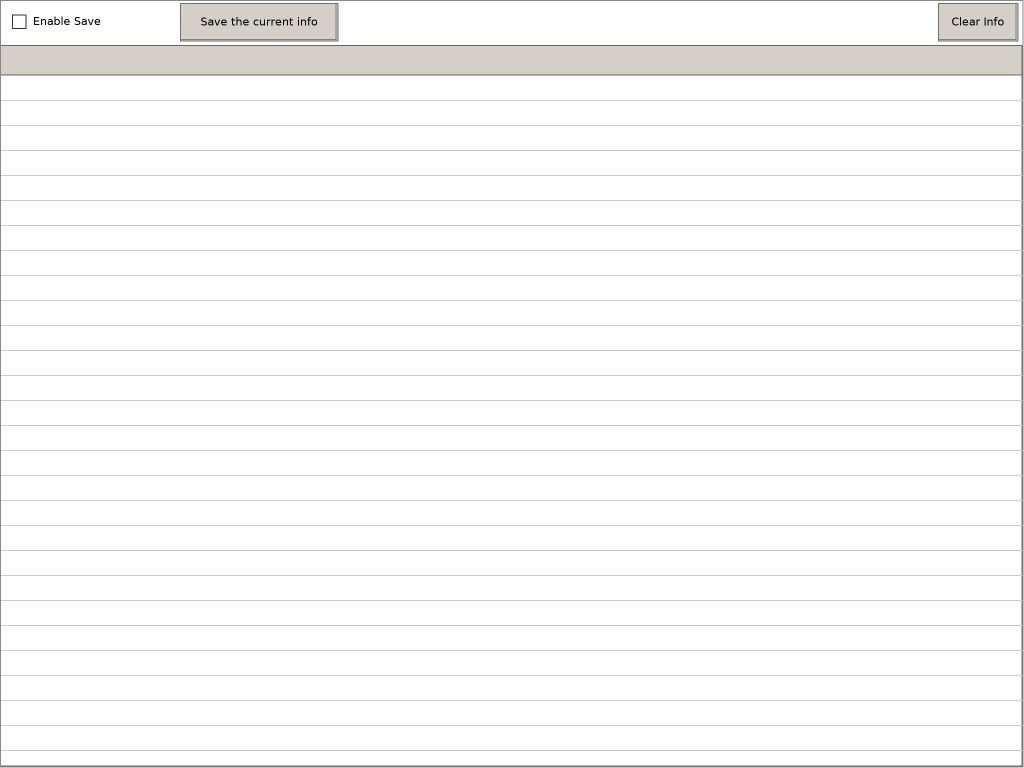
VISUALIZATION showInfo  // 1024x768
VAR_IN_OUT
	userData: printLogModule_EX_DataHMI;
END_VAR
    Checkbox (10,9 150x25), "Enable Save", variable: userData.enableSave
    Button (180,3 158x38), "Save the current info"
        tap userData.enableSaveShowLog
    Button (938,3 80x38), "Clear Info"
        tap userData.clearInformation
    Table (0,45 1022x721), data array: userData.logStrData
        p1128707560: cNumLength_showInof
        p3854506369: userData.logStrData[INDEX].sTime
        p1892666644: userData.logStrData[INDEX].msg
        p511219082: Information
END_VISUALIZATION

(* stored: Version 1.1.0.1, ProductVersion 3.1.4024.4
   Visu showInfo: Id {f1f1cc8d-65c3-4b22-82c7-cb1c47fcb084} *)
